(* PLC project MotionTest, Beckhoff Automation GmbH TwinCAT PLC Control 3.5.13.21 *)
(* stored: creationDateTime 2025-04-03T15:08:22.0993641, modificationDateTime 2025-04-03T15:08:22.1023707 *)

{attribute 'qualified_only'}
{attribute 'strict'}
TYPE MotorState :
(
    NONE        ,
    STARTING_MOTOR,
    MOVE_TO_A     ,
    MOVE_TO_B     ,
    STOPPING_MOTOR
);
END_TYPE

PROGRAM MAIN
VAR
    // ======================================================================================
    // AXIS REFERENCE
    // ======================================================================================
    // `Axis1` is a symbolic reference to a motion axis configured in the TwinCAT I/O tree.
    // It allows access to NC motion control parameters and feedback such as actual position,
    // velocity, and torque. It is passed as a parameter to motion control function blocks.
    Axis1 : AXIS_REF;

    // ======================================================================================
    // MOTION CONTROL FUNCTION BLOCKS
    // ======================================================================================
    // These blocks are part of the TwinCAT `Tc2_MC2` library and implement standard PLCopen
    // motion control functionality. They must be called cyclically and are stateful, meaning
    // they retain internal status across PLC cycles.

    // `fbPower` is responsible for powering the axis ON and OFF. It handles safety checks and
    // engages the drive when properly configured and commanded.
    fbPower : MC_Power;

    // `fbMoveA` performs an absolute positioning move to the user-defined position `posA`.
    // It is only executed when the state machine requests it.
    fbMoveA : MC_MoveAbsolute;

    // `fbMoveB` performs a second absolute move to `posB`, typically returning the axis to
    // its original or standby position.
    fbMoveB : MC_MoveAbsolute;

    // ======================================================================================
    // FSM STATE VARIABLE
    // ======================================================================================
    // `state` tracks the current execution state of the finite state machine (FSM).
    // It is based on the `MotorState` enumeration type (declared in DUTs), which should
    // define the possible states such as NONE, STARTING_MOTOR, MOVE_TO_A, etc.
    state : MotorState;

    // ======================================================================================
    // USER-DEFINED POSITION TARGETS
    // ======================================================================================
    // These are the absolute positions (in user units: e.g., mm or degrees) to which the axis
    // should move when commanded. Modify these values to configure your application’s motion
    // profile or trajectory.
    
    // `posA` is the first target point in the motion sequence. The axis will move to this
    // position after the drive is powered on.
    posA : LREAL := 100.0;

    // `posB` is the return or secondary position. The axis moves here after completing
    // the move to `posA`.
    posB : LREAL := 0.0;

    
    // ======================================================================================
    // DIGITAL I/O MAPPING
    // ======================================================================================
    // The following variables are directly mapped to physical or process image I/O.
    // TwinCAT maps `%I*` (inputs) and `%Q*` (outputs) to global process image memory.

    // `bStart` is mapped to `%I*`, meaning it corresponds to a physical or external input.
    // This allows it to be triggered by a physical button, HMI control, or another PLC task.
    // When this input is TRUE, the motion state machine begins executing.
    
    // ======================================================================================
    // START TRIGGER
    // ======================================================================================
    // `bStart` is a Boolean variable that must be set externally (e.g., from an HMI, button,
    // or test bench) to initiate the motion sequence. It acts as the FSM's entry condition.
    // The logic inside the program will automatically reset it once used.
    bStart AT%I* : BOOL := FALSE;
	

	// `bMoving` is mapped to `%Q*`, meaning it is a physical or process output variable.
    // It can be used to control an LED, HMI lamp, or any actuator to indicate that the axis
    // is currently in motion.
    bMoving AT %Q* : BOOL := FALSE;
	
    // ======================================================================================
    // AXIS FEEDBACK MONITORING
    // ======================================================================================
    // `ActPos` stores the actual position of the axis (`Axis1.NcToPlc.ActPos`).
    // This variable is updated cyclically and can be used for diagnostics, logging, visualization,
    // or condition-based decision making.
    ActPos : LREAL;
END_VAR

                  // ==========================================================================================
// === AXIS FEEDBACK ACQUISITION ===
// ==========================================================================================
//
// Read the actual position of the axis. This value is refreshed every cycle.
// Useful for display, monitoring, or control decisions.
//
ActPos := Axis1.NcToPlc.ActPos;

// Check if Axis is idle or in Motion
bMoving := state > MotorState.NONE;

// ==========================================================================================
// === FSM: STATE TRANSITIONS ===
// ==========================================================================================
//
// This block defines how the system transitions between states. Each state corresponds
// to a step in the motion sequence. Conditions must be met to advance to the next state.
//
CASE state OF

    // ---------------------------
    // IDLE STATE – Awaiting Start
    // ---------------------------
    MotorState.NONE:
        // Wait for a rising edge on `bStart`
        // This could come from an HMI, a button, or another logic block
        IF bStart THEN
            state := MotorState.STARTING_MOTOR; // Advance to motor start
            bStart := FALSE; // Reset trigger to prevent retriggering
        END_IF

    // -------------------------------------
    // STARTING MOTOR – Enable Axis Power
    // -------------------------------------
    MotorState.STARTING_MOTOR:
        // Wait for confirmation that the axis is powered
        // `Status` and `Active` must both be TRUE before moving on
        IF fbPower.Status AND fbPower.Active THEN
            state := MotorState.MOVE_TO_A;
        END_IF

    // --------------------------
    // MOVE TO POSITION A
    // --------------------------
    MotorState.MOVE_TO_A:
        // Wait until the move to position A is finished
        IF fbMoveA.Done THEN
            state := MotorState.MOVE_TO_B;
        END_IF

    // --------------------------
    // MOVE TO POSITION B
    // --------------------------
    MotorState.MOVE_TO_B:
        // Wait until the move to position B is finished
        IF fbMoveB.Done THEN
            state := MotorState.STOPPING_MOTOR;
        END_IF

    // -------------------------------------
    // STOPPING MOTOR – Disable Axis Power
    // -------------------------------------
    MotorState.STOPPING_MOTOR:
        // Confirm that the axis is no longer powered
        // When done, return to idle state
        IF NOT fbPower.Active THEN
            state := MotorState.NONE;
        END_IF

END_CASE

// ==========================================================================================
// === FSM: STATE BEHAVIOR ===
// ==========================================================================================
//
// This block defines what happens *within* each state (i.e., which function blocks
// should be executed and with what parameters). Each function block is executed
// cyclically until it completes its task.
//
CASE state OF

    // -------------------------------------
    // Enable drive power (motor ON)
    // -------------------------------------
    MotorState.STARTING_MOTOR:
        fbPower(
            Axis := Axis1,
            Enable := TRUE,           // Master enable signal
            Enable_Positive := TRUE,  // Allow positive direction motion
            Enable_Negative := TRUE   // Allow negative direction motion
        );

    // -------------------------------------
    // Send absolute move command to Position A
    // -------------------------------------
    MotorState.MOVE_TO_A:
        fbMoveA(
            Axis := Axis1,
            Execute := TRUE,           // Command the motion
            Position := posA,          // Target position (user units)
            Velocity := 50.0,          // Motion speed (user units/sec)
            Acceleration := 100.0,     // Acceleration profile
            Deceleration := 100.0      // Deceleration profile
        );

    // -------------------------------------
    // Send absolute move command to Position B
    // -------------------------------------
    MotorState.MOVE_TO_B:
        fbMoveB(
            Axis := Axis1,
            Execute := TRUE,           // Command the motion
            Position := posB,          // Target position
            Velocity := 50.0,          // Motion speed
            Acceleration := 100.0,     // Acceleration
            Deceleration := 100.0      // Deceleration
        );

    // -------------------------------------
    // Disable drive power (motor OFF)
    // -------------------------------------
    MotorState.STOPPING_MOTOR:
        fbPower(
            Axis := Axis1,
            Enable := FALSE,           // Disable drive completely
            Enable_Positive := FALSE,
            Enable_Negative := FALSE
        );

    // -------------------------------------
    // Default case – In all other states, reset function blocks
    // -------------------------------------
    ELSE
        // Important: always call MC blocks with `Execute := FALSE` when not active,
        // otherwise they may remain latched or repeat actions unnecessarily
        fbPower(
            Axis := Axis1,
            Enable := FALSE
        );

        fbMoveA(
            Axis := Axis1,
            Execute := FALSE
        );

        fbMoveB(
            Axis := Axis1,
            Execute := FALSE
        );

END_CASE

                
END_PROGRAM

CONFIGURATION Application
  RESOURCE MotionTest ON PLC
    TASK PlcTask(INTERVAL := T#0ms, PRIORITY := 20);
    PROGRAM MAIN WITH PlcTask : MAIN;
  END_RESOURCE
END_CONFIGURATION
